Staubli VAL3: s2s7En.dtx

ISO_PDU_DATA_T PDU
  [0]
    num COPT[3]
    S7telegram_T S7telegram
      [0]
        num DATA[240]
        num H[18]
    num TPKT[4]
bool bConnected
public num nAreaCT = 28
public num nAreaDB = 132
public num nAreaMK = 131
public num nAreaPA = 130
public num nAreaPE = 129
public num nAreaTM = 29
num nCC = 208
num nConnType
num nDataBuffer[500]
num nDataSize
num nErrDataRead = 768
num nErrDataWrite = 1024
num nErrISOConnFail = 6
num nErrISOInvPDU = 8
num nErrISONegPDU = 7
num nErrS7Func = 1280
num nErrTCPConnRst = 2
num nErrTCPSend = 4
num nISOPort = 102
num nISO_CR[22]
  [0] = 3
  [3] = 22
  [4] = 17
  [5] = 224
  [9] = 1
  [11] = 192
  [12] = 1
  [13] = 10
  [14] = 193
  [15] = 2
  [16] = 1
  [18] = 194
  [19] = 2
  [20] = 1
  [21] = 2
num nISOheaderSize = 7
public num nLastError
num nLastPDUType
num nLocalTSAP_HI
num nLocalTSAP_LO
num nMaxPduSize = 247
num nMinPduSize = 16
public num nNoErrors
num nPDULength
num nRDsize = 31
num nRecvTimeout = 0.5
num nRemoteTSAP_HI
num nRemoteTSAP_LO
num nS7WLCounter = 28
num nS7WLTimer = 29
num nS7_BI[37]
  [0] = 3
  [3] = 37
  [4] = 2
  [5] = 240
  [6] = 128
  [7] = 50
  [8] = 7
  [11] = 5
  [14] = 8
  [16] = 12
  [18] = 1
  [19] = 18
  [20] = 4
  [21] = 17
  [22] = 67
  [23] = 3
  [25] = 255
  [26] = 9
  [28] = 8
  [29] = 48
  [30] = 65
  [31] = 48
  [32] = 48
  [33] = 48
  [34] = 48
  [35] = 48
  [36] = 65
num nS7_PN[25]
  [0] = 3
  [3] = 25
  [4] = 2
  [5] = 240
  [6] = 128
  [7] = 50
  [8] = 1
  [11] = 4
  [14] = 8
  [17] = 240
  [20] = 1
  [22] = 1
  [24] = 240
num nS7_R[31]
  [0] = 3
  [3] = 31
  [4] = 2
  [5] = 240
  [6] = 128
  [7] = 50
  [8] = 1
  [11] = 5
  [14] = 14
  [17] = 4
  [18] = 1
  [19] = 18
  [20] = 10
  [21] = 16
  [22] = 2
  [27] = 132
num nS7_W[35]
  [0] = 3
  [3] = 31
  [4] = 2
  [5] = 240
  [6] = 128
  [7] = 50
  [8] = 1
  [11] = 5
  [14] = 14
  [17] = 4
  [18] = 1
  [19] = 18
  [20] = 10
  [21] = 16
  [22] = 2
  [27] = 132
  [32] = 4
num nShift = 17
num nTempBuffer
num nWLbit = 1
num nWLbyte = 2
num nWLcounter = 28
num nWLdword = 6
num nWLreal = 8
num nWLtimer = 29
num nWLword = 4
num nWRsize = 35
sio sioTCPclient = {link=Socket\sTcpClient}
